FUNCTION_BLOCK Pendulum4Tc
VAR_INPUT
	TimeSourceDateTime : I_PtTimesource;
END_VAR
VAR_OUTPUT
END_VAR
VAR
	_DateTime : PtDateTime;
	_Interval : PtInterval;
END_VAR


_DateTime := TimeSourceDateTime.getDateTime();

METHOD New : PtDateTime
VAR_INPUT
	Year : DINT;
	Month : DINT;
	Day : DINT;
	Hour : DINT;
	Minute : DINT;
	Second : DINT;
	Microsecond : DINT;
	TimeZone : DINT;
END_VAR
New.Set(
	Year:= Year, 
	Month:= Month, 
	Day:= Day, 
	Hour:= Hour, 
	Minute:= Minute, 
	Second:= Second, 
	Microsecond:= Microsecond, 
	TimeZone:= TimeZone);
END_METHOD

METHOD Now : PtDateTime
VAR_INPUT
END_VAR
Now := _DateTime;
END_METHOD

END_FUNCTION_BLOCK

(* stored: Version 1.1.0.1, ProductVersion 3.1.4024.12
   POU Pendulum4Tc: Id {389aeec2-3812-4b10-b54b-74a0ddd517e9}, SpecialFunc None
   Method New: Id {b29080d0-326d-4115-90bf-7e78d5b49af3}
   Method Now: Id {9ea9f490-84f7-4f1c-bd09-f76b4ad6f29b} *)
